TYPE ST_AddCommandOut :
STRUCT
	result		: REAL;
END_STRUCT
END_TYPE

(* stored: Version 1.1.0.1, ProductVersion 3.1.4022.9
   DUT ST_AddCommandOut: Id {2694872c-46f7-4930-b1f1-6309f56bc5e9} *)
